{attribute 'qualified_only'}
{attribute 'strict'}
{attribute 'to_string'}
TYPE SubTankStateEnum :
(

ready	:=	0	,//	
error	:=	100	//	


);
END_TYPE

(* stored: Version 1.1.0.1, ProductVersion 3.1.4024.11
   DUT SubTankStateEnum: Id {d330ccbf-362f-44a3-a090-0a10fa66c59c} *)
